(* IEC 61131-3 sources: std_i2980_v2.06_cp053/Source/IMM/ieccontrol/HeatingGeneral (part 2) *)

//*********************************************************************************************
// Temperature optimization
//*********************************************************************************************
//checking startconditions for temp optimization
fbRTrigRunOptimization(CLK := sv_bRunOptimization);
IF (fbRTrigRunOptimization.Q) THEN
   aCheckOptimizeStartConditions(nOptState := enOPOState);
END_IF;

IF enOPOState = enOPOState_StableFirst OR enOPOState = enOPOState_StableSecond THEN
   bGroupStable := TRUE;
   FOR i := 1 TO miNumberOfZones DO
      IF sv_ZoneArray[i].DataRetain^.bUsed THEN
         //ignore zones which are not used
         bGroupStable := bGroupStable AND (sv_ZoneArray[i].Data^.Stable = KCTRL_Stable_OK);
      END_IF;
   END_FOR;

   IF bGroupStable AND enOPOState = enOPOState_StableFirst THEN
      i := 0;
      WHILE 2*i + 1 <= miNumberOfZones DO
         IF sv_ZoneArray[2*i + 1].Data^.bSensorOK AND
            sv_ZoneArray[2*i + 1].Data^.bOutputOK AND
            sv_ZoneArray[2*i + 1].DataRetain^.SensorTypeVis <> KHW_TempSensor_none AND
            sv_ZoneArray[2*i + 1].DataRetain^.Param.opMode <> KAPPL_TempOpMode_Cooling THEN
            sv_ZoneArray[2*i + 1].Data^.bOptimize := TRUE;
            sv_ZoneArray[2*i + 1].Data^.bOptiOperatingPoint := TRUE;
         END_IF;
      i := i + 1;
      END_WHILE;
      enOPOState := enOPOState_RunFirst;
   ELSIF bGroupStable AND enOPOState = enOPOState_StableSecond THEN
      // second part of operation point calibration has to be used
      i := 1;
      WHILE 2*i <= miNumberOfZones DO
         IF sv_ZoneArray[2*i].Data^.bSensorOK AND
            sv_ZoneArray[2*i].Data^.bOutputOK AND
            sv_ZoneArray[2*i].DataRetain^.SensorTypeVis <> KHW_TempSensor_none AND
            sv_ZoneArray[2*i].DataRetain^.Param.opMode <> KAPPL_TempOpMode_Cooling THEN
            sv_ZoneArray[2*i].Data^.bOptimize := TRUE;
            sv_ZoneArray[2*i].Data^.bOptiOperatingPoint := TRUE;
         END_IF;
      i := i + 1;
      END_WHILE;
      enOPOState := enOPOState_None;
   END_IF;

END_IF;

fbRTrigOptimizationActive(CLK := sv_bOptimizationActive);//optimization started detection
fbFTrigOptimizationActive(CLK := sv_bOptimizationActive);//optimization ready detection
fbFTrigOptimizationInterrupt(CLK:= sv_bRunOptimization);//optimization stopped manually
bGroupOn := bHeatingOn;
IF fbFTrigOptimizationActive.Q THEN
   FOR i := 1 TO miNumberOfZones DO
      sv_ZoneArray[i].Data^.bOptimize := FALSE;
      // check parameters valid
      aCheckPIDParameter(iIndex2Check := i,
                         iMaxNoZones := miNumberOfZones);
   END_FOR;
   IF enOPOState = enOPOState_None THEN
      // optimization ready
      sv_bRunOptimization := FALSE;
   ELSE
      IF miNumberOfZones > 1 THEN
         enOPOState := enOPOState_StableSecond;
      ELSE  // only 1 zone optimization ready
         enOPOState := enOPOState_None;
         sv_bRunOptimization := FALSE;
      END_IF;
   END_IF;
END_IF;

//*********************************************************************************************
// Calculate set value for normal and group heating
//*********************************************************************************************
IF bHeatingOn THEN
   //call group block

   // Find Min/Max from ActValues for starting with temperatures
   // in toleranceband, checking whether the temperatures are
   // stabil relatively to each other
   MinActValues := 1000.0;
   MaxActValues := 0.0;
   FOR i := 1 TO miNumberOfZones DO
      IF sv_ZoneArray[i].Data^.bSensorOK THEN
        IF sv_ZoneArray[i].Data^.prActTemp^ < MinActValues
            AND sv_ZoneArray[i].DataRetain^.Param.bZoneUsedForGroupHeating THEN
            MinActValues := sv_ZoneArray[i].Data^.prActTemp^;
            iIndexMinZone := i;
        END_IF;
        IF sv_ZoneArray[i].Data^.prActTemp^ > MaxActValues
            AND sv_ZoneArray[i].DataRetain^.Param.bZoneUsedForGroupHeating THEN
            MaxActValues := sv_ZoneArray[i].Data^.prActTemp^;
        END_IF;
      END_IF;
   END_FOR;

   // Heating up to same temperature
   // StartGroupHeating
   IF GroupHeatingStatus = 1 THEN
      IF (((MaxActValues - MinActValues)> sv_rTolBetweenZones * 0.5) OR
          (CountStartGroupHeating < ObservationFactor)) THEN
         // Checking stability
         IF (MaxActValues - MinActValues) <= sv_rTolBetweenZones * 0.5 THEN
            CountStartGroupHeating := CountStartGroupHeating + 1;
            iIndexMinZone := 0; // no zone has set value from vis
         ELSE
            CountStartGroupHeating := 1;
         END_IF;
         IF (SetStartTemperatureGroupHeating < MinActValues) THEN
            SetStartTemperatureGroupHeating := MinActValues;
         END_IF;
         // Set the SetValues and switching of the GroupHeating temporary
         fbHeatingGroup.GroupHeating := FALSE;
          FOR i := 1 TO miNumberOfZones DO
             fbHeatingGroup.ZoneUsed[i] := sv_ZoneArray[i].DataRetain^.Param.bZoneUsedForGroupHeating;
             IF NOT sv_bKeepWarmActive THEN
                // Heating to the hotest Zonetemperature
                fbHeatingGroup.SetValues[i] := SetStartTemperatureGroupHeating;
             ELSE
                fbHeatingGroup.SetValues[i] := sv_ZoneArray[i].DataRetain^.rStandbyTempVis;
             END_IF;
             IF sv_ZoneArray[i].Data^.bSensorOK THEN
                fbHeatingGroup.ActValues[i] := sv_ZoneArray[i].Data^.prActTemp^;
             END_IF;
          END_FOR;
      ELSE
      fbHeatingGroup.GroupHeating := TRUE;
      GroupHeatingStatus := 2;
      END_IF;
   END_IF; // END GroupHeatingStatus = 1
   IF NOT (GroupHeatingStatus = 1) THEN
      FOR i := 1 TO miNumberOfZones DO
         fbHeatingGroup.ZoneUsed[i] := sv_ZoneArray[i].DataRetain^.Param.bZoneUsedForGroupHeating;
         IF NOT sv_bKeepWarmActive THEN
            IF sv_ZoneArray[i].Data^.bUseIncTemperature THEN
               fbHeatingGroup.SetValues[i] := sv_ZoneArray[i].DataRetain^.rSetValVis + sv_rIncTemperature;
            ELSE
               fbHeatingGroup.SetValues[i] := sv_ZoneArray[i].DataRetain^.rSetValVis;
            END_IF;
         ELSE
            fbHeatingGroup.SetValues[i] := sv_ZoneArray[i].DataRetain^.rStandbyTempVis;
         END_IF;
         IF sv_ZoneArray[i].Data^.bSensorOK THEN
            fbHeatingGroup.ActValues[i] := sv_ZoneArray[i].Data^.prActTemp^;
         END_IF;
      END_FOR;
      IF GroupHeatingStatus = 2 THEN
         IF (MaxActValues - MinActValues) > sv_rTolBetweenZones THEN
            bOutOfTol := TRUE;
         END_IF;
         bReadyGroupHeating := TRUE;
         FOR i := 1 TO miNumberOfZones DO
            //groupheating ignored for zones where no TI-sensor or zone not useful for GH (setter, measure mode)
            IF sv_ZoneArray[i].Data^.bSensorOK AND sv_ZoneArray[i].DataRetain^.Param.bZoneUsedForGroupHeating THEN
                IF ABS(sv_ZoneArray[i].Data^.prActTemp^-MinSetValues) > sv_rTolBetweenZones * 0.5 THEN
                    bReadyGroupHeating := FALSE;
                    EXIT;
                END_IF;
            END_IF;
         END_FOR;
         IF bReadyGroupHeating THEN
            GroupHeatingStatus := 0;
            fbHeatingGroup.GroupHeating := FALSE;
         END_IF;
      END_IF;
   END_IF;
   fbHeatingGroup(ReParam := FALSE,
                  bHeatingOn := bHeatingOn);
END_IF; //END bHeatingOn (call group block)

//*********************************************************************************************
// Set calculated set value for each zone
//*********************************************************************************************
fbRTrigSetValChanged(CLK:= fbHeatingGroup.bAnyValueChanged);
IF NOT sv_bOptimizationActive THEN
   //normal operation, copy values from group - block
   FOR i := 1 TO miNumberOfZones DO
      IF ((NOT bHeatingOn) AND (sv_ZoneArray[i].DataRetain^.Param.opMode = KAPPL_TempOpMode_Cooling)) THEN
         sv_ZoneArray[i].Data^.PWMFactor := 1.0;
         sv_ZoneArray[i].Data^.rSetVal   := sv_ZoneArray[i].DataRetain^.rSetValVis;
      ELSE
         sv_ZoneArray[i].Data^.PWMFactor := fbHeatingGroup.PWMFactor[i];
         sv_ZoneArray[i].Data^.rSetVal   := fbHeatingGroup.OutputValues[i];
      END_IF;
   END_FOR;
ELSE // optimization, use value from visualisation
    FOR i := 1 TO miNumberOfZones DO
      sv_ZoneArray[i].Data^.PWMFactor := 1.0;
      sv_ZoneArray[i].Data^.rSetVal :=  sv_ZoneArray[i].DataRetain^.rSetValVis;
   END_FOR;
END_IF;

//*********************************************************************************************
// Check state of optimization
//*********************************************************************************************
//optimization interrupted manually
IF (((fbFTrigOptimizationInterrupt.Q OR fbFTrigHeatingOn.Q) AND
     (sv_bOptimizationActive OR (enOPOState <> enOPOState_None))) OR
    (fbFTrigOptimizationInterrupt.Q AND NOT bHeatingOn AND NOT
     (sv_bOptimizationActive OR (enOPOState <> enOPOState_None)))) THEN
   FOR i := 1 TO miNumberOfZones DO
      sv_ZoneArray[i].Data^.bOptimize := FALSE;
   END_FOR;
   sv_bRunOptimization := FALSE;
END_IF;

bOptimizinActive := FALSE;
FOR i := 1 TO miNumberOfZones DO
   //check if any zone is optimizing
   IF sv_ZoneArray[i].Data^.bIsOptimizing THEN
      bOptimizinActive := TRUE;
      EXIT;
   END_IF;
END_FOR;

sv_bOptimizationActive := bOptimizinActive;

//*********************************************************************************************
// Failure control and Output
//*********************************************************************************************

//also consider zones which are not handled in groupheating
aCheckNonGroupHeatingZones();
bOtherZonesReady := aCheckNonGroupHeatingZones.bAllZonesInTolerance;

//Minutes to seconds
sv_dTempOkTimeSet :=  LINT_TO_TIME(REAL_TO_LINT(sv_rTempOkTimeSet * 60.0 * 1000.0 * 1000.0));
fbTonTempOkTime(IN := (fbHeatingGroup.AllZonesReady AND bHeatingOn AND bOtherZonesReady),
                PT := sv_dTempOkTimeSet);
sv_dTempOkTimeAct := fbTonTempOkTime.ET;
sv_rTempOkTimeAct := LINT_TO_REAL(TIME_TO_LINT(sv_dTempOkTimeAct))/(60.0 * 1000.0 * 1000.0);
bGroupTempOK := fbTonTempOkTime.Q;
fbFTrigGroupTempOK(CLK := bGroupTempOK);
fbRTrigGroupTempOK(CLK := bGroupTempOK);

// Check state of heating and set/reset alarm
// Folowing states are possible
// Heat Up Active
// Keep Warm Active
// Cool Prevent Time is running (Temperature first time in tolerance)
// None: Heating off, heating stable in operating point
IF sv_bKeepWarmActive AND NOT bKeepWarmActive THEN
    bKeepWarmActive := TRUE;
    SET_ALARM (Name := erKeepWarmActive,
                SubID1 := sv_DeviceId.CompId,
                SubID2 := sv_DeviceId.IndexId);
END_IF;
IF bKeepWarmActive AND NOT sv_bKeepWarmActive THEN
    bKeepWarmActive := FALSE;
    RESET_ALARM (Name := erKeepWarmActive,
                SubID1 := sv_DeviceId.CompId,
                SubID2 := sv_DeviceId.IndexId);
END_IF;

IF bCoolPrevent AND (bKeepWarmActive OR NOT bHeatingOn OR bGroupTempOK OR fbRTrigSetValChanged.Q) THEN
    bCoolPrevent := FALSE;
    RESET_ALARM (Name := erCoolingPrevent,
                SubID1 := sv_DeviceId.CompId,
                SubID2 := sv_DeviceId.IndexId);
END_IF;
IF NOT bCoolPrevent AND NOT bKeepWarmActive AND bHeatingOn AND NOT bGroupTempOK AND fbHeatingGroup.AllZonesReady AND bOtherZonesReady THEN
    bCoolPrevent := TRUE;
    SET_ALARM (Name := erCoolingPrevent,
                SubID1 := sv_DeviceId.CompId,
                SubID2 := sv_DeviceId.IndexId);
END_IF;

IF NOT bKeepWarmActive AND NOT mbHeatUp AND NOT bCoolPrevent AND(
    (fbRTrigHeatingOn.Q AND NOT bGroupTempOK) OR
    (bHeatingOn AND fbRTrigSetValChanged.Q AND NOT bGroupTempOK) OR
    ((sv_bGroupHeating AND fbRTrigHeatingOn.Q) OR (fbRTrigGroupHeating.Q AND bHeatingOn)) OR
    (fbFTrigOptimizationActive.Q AND NOT fbHeatingGroup.AllZonesReady)
    )THEN
    mbHeatUp := TRUE;
    SET_ALARM (Name := erHeatupActive,
                SubID1 := sv_DeviceId.CompId,
                SubID2 := sv_DeviceId.IndexId);
END_IF;
IF mbHeatUp AND (bKeepWarmActive OR bCoolPrevent OR NOT bHeatingOn OR bGroupTempOK OR fbHeatingGroup.AllZonesReady) THEN
   mbHeatUp := FALSE;
   RESET_ALARM (Name := erHeatupActive,
                SubID1 := sv_DeviceId.CompId,
                SubID2 := sv_DeviceId.IndexId);
END_IF;

(*      tolerance supervision       *)
IF fbFTrigGroupTempOK.Q THEN
    bOutOfTolerance := TRUE;
END_IF;
IF fbRTrigGroupTempOK.Q THEN
    bOutOfTolerance := FALSE;
END_IF;
IF ((bOutOfTolerance OR fbRTrigGroupTempOK.Q) AND
    (NOT (mbHeatUp OR bCoolPrevent OR sv_bRunOptimization)) OR (NOT bHeatingOn)) THEN

    FOR i := 1 TO miNumberOfZones DO
        (* searching for the zones which are out ouf tol *)
        IF (sv_ZoneArray[i].Data^.bToleranceError AND (NOT ToleranceAlarm[i])) AND
           (bHeatingOn AND (NOT (mbHeatUp OR bCoolPrevent))) THEN
            (* setting tolerance error *)
            IF ((sv_ZoneArray[i].Data^.bEmgOperation AND sv_OperationMode >= nHalfAutomatic)) OR
                bKeepWarmActive OR bGroupActive THEN
               ; // no Alarm Emergency operation mode
            ELSE
               ToleranceAlarm[i] := TRUE;
               SET_ALARM (Name := erZoneOutOfTol,
                        SubID1 := sv_DeviceId.CompId,
                        SubID2 := sv_DeviceId.IndexId,
                        SubID3 := i);
           END_IF;
        END_IF;

        IF  (NOT sv_ZoneArray[i].Data^.bToleranceError AND ToleranceAlarm[i]) OR
            (NOT bHeatingOn AND ToleranceAlarm[i]) OR (NOT sv_ZoneArray[i].DataRetain^.bUsed)  THEN

            ToleranceAlarm[i] := FALSE;
            RESET_ALARM (Name := erZoneOutOfTol,
                    SubID1 := sv_DeviceId.CompId,
                    SubID2 := sv_DeviceId.IndexId,
                    SubID3 := i);
        END_IF;
    END_FOR;
END_IF;

// set/reset status message during temp.optimization
IF fbRTrigOptimizationActive.Q THEN
    SET_ALARM (Name := erOptimizationActive,
              SubID1 := sv_DeviceId.CompId,
              SubID2 := sv_DeviceId.IndexId);
END_IF;

IF fbFTrigOptimizationActive.Q THEN
    RESET_ALARM (Name := erOptimizationActive,
                SubID1 := sv_DeviceId.CompId,
                SubID2 := sv_DeviceId.IndexId);
END_IF;

fbRTrigOutOfTol(CLK:=bOutOfTol);
IF fbRTrigOutOfTol.Q THEN
   SET_ALARM (Name := erOutOfTol,
              SubID1 := sv_DeviceId.CompId,
              SubID2 := sv_DeviceId.IndexId);
END_IF;

bGroupActive := (GroupHeatingStatus > 0);

@END_Body

@@@BEG_Comment@@@
@TL(0)

@@@END_Comment@@@

@BEG_Body
@TL(9)
(**************************************** WARNING ********************************************
 *** The KEBA Kemro K2 System including software is not intended for safety control tasks! ***
 ***                       For further information see Comment tab!                        ***
 *********************************************************************************************)

//reparam Group
mbInit := FALSE;
sv_bReParamGroup := FALSE;

@END_Body

@@@BEG_Comment@@@
@TL(0)

@@@END_Comment@@@

@BEG_Body
@TL(7)
(**************************************** WARNING ********************************************
 *** The KEBA Kemro K2 System including software is not intended for safety control tasks! ***
 ***                       For further information see Comment tab!                        ***
 *********************************************************************************************)

START_PROCESS_ALGORITHM(paCheckNumberOfZones);

@END_Body

@@@BEG_Comment@@@
@TL(0)

@@@END_Comment@@@

@BEG_Body
@TL(52)
(**************************************** WARNING ********************************************
 *** The KEBA Kemro K2 System including software is not intended for safety control tasks! ***
 ***                       For further information see Comment tab!                        ***
 *********************************************************************************************)

IF mbInitDone THEN

   FOR i := 1 TO sv_iMaxNumberOfZones DO

      IF i <= sv_iZonesAvailable AND i <= sv_iNumberOfZones AND sv_ZoneArray[i].bLinked THEN
            //tell the zone that it will be used
            //set counter for aRun to prevent from nullpointerexception if wrong mold data was loaded (sv_iNumberOfZones > sv_iZonesAvailable)
            miNumberOfZones := i;
            // Dont set value higher than max allowed temperature
            sv_ZoneArray[i].Data^.bOutputNotAllowed := FALSE;
            sv_ZoneArray[i].DataRetain^.rSetValVis := MIN(sv_rMaxTemperature, sv_ZoneArray[i].DataRetain^.rSetValVis);
            // heating nozzle zone is always used
            IF NOT (sv_ZoneArray[i].DataRetain^.bIsHotrunner OR sv_ZoneArray[i].DataRetain^.ZoneType = enZoneTypeBlock) THEN
               sv_ZoneArray[i].DataRetain^.bUsed := TRUE;
            END_IF;
      ELSIF sv_ZoneArray[i].bLinked THEN
            sv_ZoneArray[i].DataRetain^.bUsed := FALSE;
      END_IF;

      IF i > sv_iZonesAvailable AND i <= sv_iNumberOfZones THEN
         //zone is used but Hardware is not OK -> error
            SET_ALARM(Name := erZoneNotAvailable,
                      SubID1 := sv_DeviceId.CompId,
                      SubID2 := sv_DeviceId.IndexId,
                      SubID3 := i);
      END_IF;

      IF  i > sv_iNumberOfZones AND i <= iNumberOfZonesOld AND i > sv_iZonesAvailable THEN
         //reset alarm if sv_iNumberOfZones has been reduced
         RESET_ALARM(Name := erZoneNotAvailable,
                     SubID1 := sv_DeviceId.CompId,
                     SubID2 := sv_DeviceId.IndexId,
                     SubID3 := i);
         IF (sv_ZoneArray[i].bLinked) AND
            NOT (sv_ZoneArray[i].DataRetain^.bIsHotrunner OR sv_ZoneArray[i].DataRetain^.ZoneType = enZoneTypeBlock) THEN
            sv_ZoneArray[i].DataRetain^.bUsed := TRUE;
         END_IF;

      END_IF;
   END_FOR;
   STOP_PROCESS_ALGORITHM();
END_IF;

iNumberOfZonesOld := sv_iNumberOfZones;

@END_Body

@@@BEG_Comment@@@
@TL(0)

@@@END_Comment@@@

@BEG_Body
@TL(7)
// After max temperature changed, dont allow higher set values
FOR i := 1 TO miNumberOfZones DO
    IF sv_ZoneArray[i].DataRetain^.rSetValVis > sv_rMaxTemperature THEN
       sv_ZoneArray[i].DataRetain^.rSetValVis := sv_rMaxTemperature;
    END_IF;
END_FOR;

@END_Body

@@@BEG_Comment@@@
@TL(0)

@@@END_Comment@@@

@BEG_Body
@TL(18)
IF sv_bUndoChangeHeatingParams THEN
   IF NOT mbInitDone THEN
      sv_bUndoChangeHeatingParams := FALSE;
      RETURN;
   END_IF;
   FOR i := 1 TO miNumberOfZones DO
      IF sv_ZoneArray[i].DataRetain^.Param.bOldPIDAvailable THEN
         sv_ZoneArray[i].DataRetain^.Param.pidParam := sv_ZoneArray[i].DataRetain^.Param.pidParamLastOpt;
         sv_bUsePidOP := FALSE;
         sv_bReParamGroup := TRUE;
         sv_ZoneArray[i].DataRetain^.Param.bOldPIDAvailable := FALSE;
      END_IF;
   END_FOR;
   //reparam tempgroup
   // reset sv
   sv_bUndoChangeHeatingParams := FALSE;
END_IF;

@END_Body

@@@BEG_Comment@@@
@TL(0)

@@@END_Comment@@@

@BEG_Body
@TL(7)
(**************************************** WARNING ********************************************
 *** The KEBA Kemro K2 System including software is not intended for safety control tasks! ***
 ***                       For further information see Comment tab!                        ***
 *********************************************************************************************)

rActTemp := sv_ZoneArray[miLeadingZone].Data^.prActTemp^;

@END_Body

@@@BEG_Comment@@@
@TL(0)

@@@END_Comment@@@
@END_Body

@END_Contents

(* ---- ABHopperCooling.pu ---- *)
(*
This Algorithm Block is responsible for
  - hopper temp. supervision
  - hopper cooling

*)

IMPORT_OVER_LISTFILE
 KSWO_AddVariable
, SET_ALARM
, RESET_ALARM
, FGetHWPath
, GET_MY_FU_NAME
, KHW_TempSensor
, tsDeviceId
, KSWO_Status
, R_TRIG

END_IMPORT

ALGORITHM_BLOCK ABHopperCooling #DUMMY_EDIT_BLOCK

SYSTEM_VAR
 do_HopperCooler : BOOL;
 ti_HopperTemp : REAL;
 ti_HopperTemp_sensor : KHW_TempSensor;
 ti_HopperTemp_stat : BOOL;
 sv_rTempStartCooling : REAL (* start cooling at this temperature *);
 sv_rTempStopCooling : REAL (* stop cooling at this temperature *);
 sv_rWarnTemp : REAL (* a warning is displayed if hopper temperature increases this value *);
 sv_rAlarmTemp : REAL (* an alarm is displayed if hopper temperature increases this value *);
 sv_HopperTempSensorType : KHW_TempSensor (* sensor type *);
 sv_rHopperTempHysteresis : REAL;
 sv_DeviceId : tsDeviceId;
END_VAR

SYSTEM_OBJECT
 PU_Task_7 : TASK;
 TaskSlow : TASK;
 erHopperTempWarning : ALARM;
 erHopperTempTooHigh : ALARM;
 erHopperTempSensor : ALARM;
END_OBJECT

VAR
 mbSensorError : BOOL;
 msHWPath : STRING(255);
 mpbSensorState : REFTO BOOL;
END_VAR

ALGORITHM aSensorState

#BEGIN_EDIT_BLOCK
(**************************************** WARNING ********************************************
 *** The KEBA Kemro K2 System including software is not intended for safety control tasks! ***
 ***                       For further information see Comment tab!                        ***
 *********************************************************************************************)

mbSensorError := ti_HopperTemp_stat;

IF mbSensorError THEN

   //reset digital output for cooling in case of sensor error
   IF IS_LINKED(do_HopperCooler) THEN
      do_HopperCooler := FALSE;
   END_IF;

   SET_ALARM(Name := erHopperTempSensor,
             SubID1 := sv_DeviceId.CompId,
             SubID2 := sv_DeviceId.IndexId,
             Param1 := msHWPath);
ELSE
   RESET_ALARM(Name := erHopperTempSensor,
               SubID1 := sv_DeviceId.CompId,
               SubID2 := sv_DeviceId.IndexId);
END_IF;

;#END_EDIT_BLOCK END_ALGORITHM

(*
Check which Inputs and Outputs are available and start according process algorithms
*)

PROCESS_ALGORITHM paInit ON TaskSlow AUTOSTART

VAR
 swoState : KSWO_Status;
END_VAR
#BEGIN_EDIT_BLOCK
(**************************************** WARNING ********************************************
 *** The KEBA Kemro K2 System including software is not intended for safety control tasks! ***
 ***                       For further information see Comment tab!                        ***
 *********************************************************************************************)

IF IS_LINKED(ti_HopperTemp) AND IS_LINKED(ti_HopperTemp_stat) THEN

   ti_HopperTemp_sensor := sv_HopperTempSensorType;

   msHWPath := FGetHWPath(CONCAT(GET_MY_FU_NAME(),'.ti_HopperTemp'), TRUE);
   mpbSensorState := @ti_HopperTemp_stat;

   aSensorState();

   swoState := KSWO_AddVariable( Task := TaskSlow,
                                 Name := 'HopperTemperature',
                                 Variable := ti_HopperTemp);

   //start supervision of hopper temperature
   START_PROCESS_ALGORITHM(paHopperTempSupervision);

   IF IS_LINKED(do_HopperCooler) THEN
      //start algorithm for hopper cooling
      START_PROCESS_ALGORITHM(paHopperCooler);
   END_IF;
END_IF;

STOP_PROCESS_ALGORITHM();

;#END_EDIT_BLOCK END_ALGORITHM

(*
In this algorithm the supervision of the material temperature is done.
If actual material temp is higher than the alarm temperature an alarm is set.
If actual material temperature is lower than alarm temp -5° the alarm is resetted.
Setting the material temp high - alarm causes a stop of the motor!
Switching on the motor is only possible if the material temperature is ok again.
*)

PROCESS_ALGORITHM paHopperTempSupervision ON TaskSlow

VAR
 fbRTrigWarningTemp : R_TRIG;
 fbRTrigAlarmTemp : R_TRIG;
 fbRTrigWarningTempOk : R_TRIG;
 fbRTrigAlarmTempOk : R_TRIG;
END_VAR
#BEGIN_EDIT_BLOCK
(**************************************** WARNING ********************************************
 *** The KEBA Kemro K2 System including software is not intended for safety control tasks! ***
 ***                       For further information see Comment tab!                        ***
 *********************************************************************************************)

fbRTrigWarningTemp(CLK := (ti_HopperTemp > sv_rWarnTemp));
fbRTrigWarningTempOk(CLK := (ti_HopperTemp < (sv_rWarnTemp - sv_rHopperTempHysteresis)));

fbRTrigAlarmTemp(CLK := (ti_HopperTemp > sv_rAlarmTemp));
fbRTrigAlarmTempOk(CLK := (ti_HopperTemp < (sv_rAlarmTemp - sv_rHopperTempHysteresis)));

IF fbRTrigWarningTemp.Q THEN
   //set alarm if warning temp is exceeded
   SET_ALARM (Name := erHopperTempWarning,
              SubID1 := sv_DeviceId.CompId,
              SubID2 := sv_DeviceId.IndexId);
END_IF;

IF fbRTrigWarningTempOk.Q THEN
   //reset alarm if temp is ok again
   RESET_ALARM (Name := erHopperTempWarning,
                SubID1 := sv_DeviceId.CompId,
                SubID2 := sv_DeviceId.IndexId);
END_IF;

IF fbRTrigAlarmTemp.Q THEN
   //set alarm if alarm temp is exceeded
   SET_ALARM (Name := erHopperTempTooHigh,
              SubID1 := sv_DeviceId.CompId,
              SubID2 := sv_DeviceId.IndexId);
END_IF;

IF fbRTrigAlarmTempOk.Q THEN
   //set alarm if temp is ok again
   RESET_ALARM (Name := erHopperTempTooHigh,
                SubID1 := sv_DeviceId.CompId,
                SubID2 := sv_DeviceId.IndexId);
END_IF;

;#END_EDIT_BLOCK END_ALGORITHM

(*
If a digital output for hopper cooling is available it will be set if the
actual material temperature is higher than start cooling temperature.
The DO will be resetted after the actual temperature is lower than stop cooling temperature.
In case of a sensor error the DO will also be resetted.
*)

PROCESS_ALGORITHM paHopperCooler ON TaskSlow

VAR
 fbRTrigStartCooling : R_TRIG;
 fbRTrigStopCooling : R_TRIG;
END_VAR
#BEGIN_EDIT_BLOCK
(**************************************** WARNING ********************************************
 *** The KEBA Kemro K2 System including software is not intended for safety control tasks! ***
 ***                       For further information see Comment tab!                        ***
 *********************************************************************************************)

fbRTrigStartCooling(CLK := (ti_HopperTemp > sv_rTempStartCooling));
fbRTrigStopCooling(CLK := (ti_HopperTemp < sv_rTempStopCooling));

IF fbRTrigStartCooling.Q AND NOT mbSensorError THEN
   //set digital output for cooling
   do_HopperCooler := TRUE;
END_IF;

IF fbRTrigStopCooling.Q THEN
   //reset digital output for cooling
   do_HopperCooler := FALSE;
END_IF;

;#END_EDIT_BLOCK END_ALGORITHM

POSTUPDATE_ALGORITHM pSensorTypeChanged ON PU_Task_7 WITH sv_HopperTempSensorType

#BEGIN_EDIT_BLOCK
(**************************************** WARNING ********************************************
 *** The KEBA Kemro K2 System including software is not intended for safety control tasks! ***
 ***                       For further information see Comment tab!                        ***
 *********************************************************************************************)

//copy selected sensor type
ti_HopperTemp_sensor := sv_HopperTempSensorType;

;#END_EDIT_BLOCK END_ALGORITHM

(*
react on changes of material temp sensor state
*)

POSTUPDATE_ALGORITHM pSensorStateChanged ON PU_Task_7 WITH mpbSensorState^

#BEGIN_EDIT_BLOCK
(**************************************** WARNING ********************************************
 *** The KEBA Kemro K2 System including software is not intended for safety control tasks! ***
 ***                       For further information see Comment tab!                        ***
 *********************************************************************************************)

aSensorState();

;#END_EDIT_BLOCK END_ALGORITHM

END_ALGORITHM_BLOCK

#END_OF_IEC_PART

@Puma @IecEditor 6 68 @Pou 25
@@@BEG_Comment@@@
This Algorithm Block is responsible for
  - hopper temp. supervision
  - hopper cooling

@@@END_Comment@@@

@BEG_Contents

@BEG_Func
@RT(17)FuncTreeContainer
5
@Var @RT(16)KSWO_AddVariable @RT(0) @T @T @DERIVED 0 @F @RT(22)KEBA_STANDARD_FUNCTION @F
@T
@BEG_Attrib
0 @RT(0) @RT(0)
@END_Attrib
1 1 @F @F @F @F

@Var @RT(9)SET_ALARM @RT(0) @T @T @DERIVED 0 @F @RT(23)KEBA_STANDARD_PROCEDURE @F
@T
@BEG_Attrib
0 @RT(0) @RT(0)
@END_Attrib
1 1 @F @F @F @F

@Var @RT(11)RESET_ALARM @RT(0) @T @T @DERIVED 0 @F @RT(23)KEBA_STANDARD_PROCEDURE @F
@T
@BEG_Attrib
0 @RT(0) @RT(0)
@END_Attrib
1 1 @F @F @F @F

@Var @RT(10)FGetHWPath @RT(0) @T @T @DERIVED 0 @F @RT(8)FUNCTION @F
@T
@BEG_Attrib
0 @RT(0) @RT(0)
@END_Attrib
1 1 @F @F @F @F

@Var @RT(14)GET_MY_FU_NAME @RT(0) @T @T @DERIVED 0 @F @RT(22)KEBA_STANDARD_FUNCTION @F
@T
@BEG_Attrib
0 @RT(0) @RT(0)
@END_Attrib
1 1 @F @F @F @F

@END_Func

@BEG_Const
@RT(18)ConstTreeContainer
0
@END_Const

@BEG_Export

@BEG_Kind
@ALGORITHM_BLOCK @RT(15)ABHopperCooling @STRUCTURED_TEXT
@RT(0) @RT(0) @RT(0)
@END_Kind

@BEG_Dcl
@RT(16)DclTreeContainer
19
@Var @RT(15)do_HopperCooler @RT(0) @T @F @DT @RT(4)BOOL @RT(0) @T @T @BASIC 0 @F
@F @F
@T
@BEG_Attrib
3 @RT(0) @RT(0) @RT(0)
@END_Attrib
1 8 @F @F @F @F

@Var @RT(13)ti_HopperTemp @RT(0) @T @F @DT @RT(4)REAL @RT(0) @T @T @BASIC 0 @F
@F @F
@T
@BEG_Attrib
3 @RT(0) @RT(0) @RT(0)
@END_Attrib
1 8 @F @F @F @F

@Var @RT(20)ti_HopperTemp_sensor @RT(0) @T @T @DERIVED 0 @T @T @DT @RT(14)KHW_TempSensor @RT(0) @T @T @UNKNOWN 0 @F
@F @F
@T
@BEG_Attrib
3 @RT(0) @RT(0) @RT(0)
@END_Attrib
1 8 @F @F @F @F

@Var @RT(18)ti_HopperTemp_stat @RT(0) @T @F @DT @RT(4)BOOL @RT(0) @T @T @BASIC 0 @F
@F @F
@T
@BEG_Attrib
3 @RT(0) @RT(0) @RT(0)
@END_Attrib
1 8 @F @F @F @F

@Var @RT(20)sv_rTempStartCooling @RT(0) @T @F @DT @RT(4)REAL @RT(0) @T @T @BASIC 0 @F
@F @F
@T
@BEG_Attrib
3 @RT(0) @RT(33)start cooling at this temperature @RT(0)
@END_Attrib
1 8 @F @F @F @F

@Var @RT(19)sv_rTempStopCooling @RT(0) @T @F @DT @RT(4)REAL @RT(0) @T @T @BASIC 0 @F
@F @F
@T
@BEG_Attrib
3 @RT(0) @RT(32)stop cooling at this temperature @RT(0)
@END_Attrib
1 8 @F @F @F @F

@Var @RT(12)sv_rWarnTemp @RT(0) @T @F @DT @RT(4)REAL @RT(0) @T @T @BASIC 0 @F
@F @F
@T
@BEG_Attrib
3 @RT(0) @RT(65)a warning is displayed if hopper temperature increases this value @RT(0)
@END_Attrib
1 8 @F @F @F @F

@Var @RT(13)sv_rAlarmTemp @RT(0) @T @F @DT @RT(4)REAL @RT(0) @T @T @BASIC 0 @F
@F @F
@T
@BEG_Attrib
3 @RT(0) @RT(64)an alarm is displayed if hopper temperature increases this value @RT(0)
@END_Attrib
1 8 @F @F @F @F

@Var @RT(23)sv_HopperTempSensorType @RT(0) @T @T @DERIVED 0 @T @T @DT @RT(14)KHW_TempSensor @RT(0) @T @T @UNKNOWN 0 @F
@F @F
@T
@BEG_Attrib
3 @RT(0) @RT(11)sensor type @RT(0)
@END_Attrib
1 8 @F @F @F @F

@Var @RT(9)PU_Task_7 @RT(0) @T @F @DT @RT(4)TASK @RT(0) @T @T @BASIC 0 @F
@F @F
@T
@BEG_Attrib
3 @RT(0) @RT(0) @RT(0)
@END_Attrib
1 7 @F @F @F @F

@Var @RT(8)TaskSlow @RT(0) @T @F @DT @RT(4)TASK @RT(0) @T @T @BASIC 0 @F
@F @F
@T
@BEG_Attrib
3 @RT(0) @RT(0) @RT(0)
@END_Attrib
1 7 @F @F @F @F

@Var @RT(19)erHopperTempWarning @RT(0) @T @F @DT @RT(5)ALARM @RT(0) @T @T @BASIC 0 @F
@F @F
@T
@BEG_Attrib
3 @RT(0) @RT(0) @RT(0)
@END_Attrib
1 7 @F @F @F @F

@Var @RT(19)erHopperTempTooHigh @RT(0) @T @F @DT @RT(5)ALARM @RT(0) @T @T @BASIC 0 @F
@F @F
@T
@BEG_Attrib
3 @RT(0) @RT(0) @RT(0)
@END_Attrib
1 7 @F @F @F @F

@Var @RT(18)erHopperTempSensor @RT(0) @T @F @DT @RT(5)ALARM @RT(0) @T @T @BASIC 0 @F
@F @F
@T
@BEG_Attrib
3 @RT(0) @RT(0) @RT(0)
@END_Attrib
1 7 @F @F @F @F

@Var @RT(13)mbSensorError @RT(0) @T @F @DT @RT(4)BOOL @RT(0) @T @T @BASIC 0 @F
@F @F
@T
@BEG_Attrib
3 @RT(0) @RT(0) @RT(0)
@END_Attrib
1 0 @F @F @F @F

@Var @RT(24)sv_rHopperTempHysteresis @RT(0) @T @F @DT @RT(4)REAL @RT(0) @T @T @BASIC 0 @F
@F @F
@T
@BEG_Attrib
3 @RT(0) @RT(0) @RT(0)
@END_Attrib
1 8 @F @F @F @F

@Var @RT(8)msHWPath @RT(0) @T @F @DT @RT(11)STRING(255) @RT(0) @T @T @STRING 0 @F @RT(3)255 @F
@F @F
@T
@BEG_Attrib
3 @RT(0) @RT(0) @RT(0)
@END_Attrib
1 0 @F @F @F @F

@Var @RT(14)mpbSensorState @RT(0) @T @T @REFTO 0 @T @DT @RT(4)BOOL @RT(0) @T @T @BASIC 0 @F
@F @F
@T
@BEG_Attrib
3 @RT(0) @RT(0) @RT(0)
@END_Attrib
1 0 @F @F @F @F

@Var @RT(11)sv_DeviceId @RT(0) @T @T @DERIVED 0 @F @RT(10)tsDeviceId @F
@T
@BEG_Attrib
3 @RT(0) @RT(0) @RT(0)
@END_Attrib
1 8 @F @F @F @F

@END_Dcl

@END_Export

@BEG_Body

6

@BEG_Export

@BEG_Algo
@ALGORITHM @RT(12)aSensorState @STRUCTURED_TEXT
@RT(0) @RT(0) @RT(0) @F @F
@END_Algo

@BEG_Dcl
@RT(16)DclTreeContainer
0
@END_Dcl

@END_Export

@BEG_Export

@BEG_Algo
@PROCESS_ALGORITHM @RT(6)paInit @STRUCTURED_TEXT
@RT(0) @RT(0) @RT(8)TaskSlow @T @F
@END_Algo

@BEG_Dcl
@RT(16)DclTreeContainer
1
@Var @RT(8)swoState @RT(0) @T @T @DERIVED 0 @T @T @DT @RT(11)KSWO_Status @RT(0) @T @T @UNKNOWN 0 @F
@F @F
@T
@BEG_Attrib
3 @RT(0) @RT(0) @RT(0)
@END_Attrib
1 0 @F @F @F @F

@END_Dcl

@END_Export

@BEG_Export

@BEG_Algo
@PROCESS_ALGORITHM @RT(23)paHopperTempSupervision @STRUCTURED_TEXT
@RT(0) @RT(0) @RT(8)TaskSlow @F @F
@END_Algo

@BEG_Dcl
@RT(16)DclTreeContainer
4
@Var @RT(18)fbRTrigWarningTemp @RT(0) @T @T @DERIVED 0 @T @T @DT @RT(6)R_TRIG @RT(0) @T @T @UNKNOWN 0 @F
@F @F
@T
@BEG_Attrib
3 @RT(0) @RT(0) @RT(0)
@END_Attrib
1 0 @F @F @F @F

@Var @RT(16)fbRTrigAlarmTemp @RT(0) @T @T @DERIVED 0 @T @T @DT @RT(6)R_TRIG @RT(0) @T @T @UNKNOWN 0 @F
@F @F
@T
@BEG_Attrib
3 @RT(0) @RT(0) @RT(0)
@END_Attrib
1 0 @F @F @F @F

@Var @RT(20)fbRTrigWarningTempOk @RT(0) @T @T @DERIVED 0 @T @T @DT @RT(6)R_TRIG @RT(0) @T @T @UNKNOWN 0 @F
@F @F
@T
@BEG_Attrib
3 @RT(0) @RT(0) @RT(0)
@END_Attrib
1 0 @F @F @F @F

@Var @RT(18)fbRTrigAlarmTempOk @RT(0) @T @T @DERIVED 0 @T @T @DT @RT(6)R_TRIG @RT(0) @T @T @UNKNOWN 0 @F
@F @F
@T
@BEG_Attrib
3 @RT(0) @RT(0) @RT(0)
@END_Attrib
1 0 @F @F @F @F

@END_Dcl

@END_Export

@BEG_Export

@BEG_Algo
@PROCESS_ALGORITHM @RT(14)paHopperCooler @STRUCTURED_TEXT
@RT(0) @RT(0) @RT(8)TaskSlow @F @F
@END_Algo

@BEG_Dcl
@RT(16)DclTreeContainer
2
@Var @RT(19)fbRTrigStartCooling @RT(0) @T @T @DERIVED 0 @T @T @DT @RT(6)R_TRIG @RT(0) @T @T @UNKNOWN 0 @F
@F @F
@T
@BEG_Attrib
3 @RT(0) @RT(0) @RT(0)
@END_Attrib
1 0 @F @F @F @F

@Var @RT(18)fbRTrigStopCooling @RT(0) @T @T @DERIVED 0 @T @T @DT @RT(6)R_TRIG @RT(0) @T @T @UNKNOWN 0 @F
@F @F
@T
@BEG_Attrib
3 @RT(0) @RT(0) @RT(0)
@END_Attrib
1 0 @F @F @F @F

@END_Dcl

@END_Export

@BEG_Export

@BEG_Algo
@POSTUPDATE_ALGORITHM @RT(18)pSensorTypeChanged @STRUCTURED_TEXT
@RT(0) @RT(23)sv_HopperTempSensorType @RT(9)PU_Task_7 @F @F
@END_Algo

@BEG_Dcl
@RT(16)DclTreeContainer
0
@END_Dcl

@END_Export

@BEG_Export

@BEG_Algo
@POSTUPDATE_ALGORITHM @RT(19)pSensorStateChanged @STRUCTURED_TEXT
@RT(0) @RT(15)mpbSensorState^ @RT(9)PU_Task_7 @F @F
@END_Algo

@BEG_Dcl
@RT(16)DclTreeContainer
0
@END_Dcl

@END_Export

@BEG_Body
@TL(24)
(**************************************** WARNING ********************************************
 *** The KEBA Kemro K2 System including software is not intended for safety control tasks! ***
 ***                       For further information see Comment tab!                        ***
 *********************************************************************************************)

mbSensorError := ti_HopperTemp_stat;

IF mbSensorError THEN

   //reset digital output for cooling in case of sensor error
   IF IS_LINKED(do_HopperCooler) THEN
      do_HopperCooler := FALSE;
   END_IF;

   SET_ALARM(Name := erHopperTempSensor,
             SubID1 := sv_DeviceId.CompId,
             SubID2 := sv_DeviceId.IndexId,
             Param1 := msHWPath);
ELSE
   RESET_ALARM(Name := erHopperTempSensor,
               SubID1 := sv_DeviceId.CompId,
               SubID2 := sv_DeviceId.IndexId);
END_IF;

@END_Body

@@@BEG_Comment@@@
@TL(0)

@@@END_Comment@@@

@BEG_Body
@TL(30)
(**************************************** WARNING ********************************************
 *** The KEBA Kemro K2 System including software is not intended for safety control tasks! ***
 ***                       For further information see Comment tab!                        ***
 *********************************************************************************************)

IF IS_LINKED(ti_HopperTemp) AND IS_LINKED(ti_HopperTemp_stat) THEN

   ti_HopperTemp_sensor := sv_HopperTempSensorType;

   msHWPath := FGetHWPath(CONCAT(GET_MY_FU_NAME(),'.ti_HopperTemp'), TRUE);
   mpbSensorState := @ti_HopperTemp_stat;

   aSensorState();

   swoState := KSWO_AddVariable( Task := TaskSlow,
                                 Name := 'HopperTemperature',
                                 Variable := ti_HopperTemp);

   //start supervision of hopper temperature
   START_PROCESS_ALGORITHM(paHopperTempSupervision);

   IF IS_LINKED(do_HopperCooler) THEN
      //start algorithm for hopper cooling
      START_PROCESS_ALGORITHM(paHopperCooler);
   END_IF;
END_IF;

STOP_PROCESS_ALGORITHM();

@END_Body

@@@BEG_Comment@@@
@TL(1)
Check which Inputs and Outputs are available and start according process algorithms
@@@END_Comment@@@

@BEG_Body
@TL(39)
(**************************************** WARNING ********************************************
 *** The KEBA Kemro K2 System including software is not intended for safety control tasks! ***
 ***                       For further information see Comment tab!                        ***
 *********************************************************************************************)

fbRTrigWarningTemp(CLK := (ti_HopperTemp > sv_rWarnTemp));
fbRTrigWarningTempOk(CLK := (ti_HopperTemp < (sv_rWarnTemp - sv_rHopperTempHysteresis)));

fbRTrigAlarmTemp(CLK := (ti_HopperTemp > sv_rAlarmTemp));
fbRTrigAlarmTempOk(CLK := (ti_HopperTemp < (sv_rAlarmTemp - sv_rHopperTempHysteresis)));

IF fbRTrigWarningTemp.Q THEN
   //set alarm if warning temp is exceeded
   SET_ALARM (Name := erHopperTempWarning,
              SubID1 := sv_DeviceId.CompId,
              SubID2 := sv_DeviceId.IndexId);
END_IF;

IF fbRTrigWarningTempOk.Q THEN
   //reset alarm if temp is ok again
   RESET_ALARM (Name := erHopperTempWarning,
                SubID1 := sv_DeviceId.CompId,
                SubID2 := sv_DeviceId.IndexId);
END_IF;

IF fbRTrigAlarmTemp.Q THEN
   //set alarm if alarm temp is exceeded
   SET_ALARM (Name := erHopperTempTooHigh,
              SubID1 := sv_DeviceId.CompId,
              SubID2 := sv_DeviceId.IndexId);
END_IF;

IF fbRTrigAlarmTempOk.Q THEN
   //set alarm if temp is ok again
   RESET_ALARM (Name := erHopperTempTooHigh,
                SubID1 := sv_DeviceId.CompId,
                SubID2 := sv_DeviceId.IndexId);
END_IF;

@END_Body

@@@BEG_Comment@@@
@TL(5)
In this algorithm the supervision of the material temperature is done.
If actual material temp is higher than the alarm temperature an alarm is set.
If actual material temperature is lower than alarm temp -5° the alarm is resetted.
Setting the material temp high - alarm causes a stop of the motor!
Switching on the motor is only possible if the material temperature is ok again.
@@@END_Comment@@@

@BEG_Body
@TL(20)
(**************************************** WARNING ********************************************
 *** The KEBA Kemro K2 System including software is not intended for safety control tasks! ***
 ***                       For further information see Comment tab!                        ***
 *********************************************************************************************)

fbRTrigStartCooling(CLK := (ti_HopperTemp > sv_rTempStartCooling));
fbRTrigStopCooling(CLK := (ti_HopperTemp < sv_rTempStopCooling));

IF fbRTrigStartCooling.Q AND NOT mbSensorError THEN
   //set digital output for cooling
   do_HopperCooler := TRUE;
END_IF;

IF fbRTrigStopCooling.Q THEN
   //reset digital output for cooling
   do_HopperCooler := FALSE;
END_IF;

@END_Body

@@@BEG_Comment@@@
@TL(4)
If a digital output for hopper cooling is available it will be set if the
actual material temperature is higher than start cooling temperature.
The DO will be resetted after the actual temperature is lower than stop cooling temperature.
In case of a sensor error the DO will also be resetted.
@@@END_Comment@@@

@BEG_Body
@TL(9)
(**************************************** WARNING ********************************************
 *** The KEBA Kemro K2 System including software is not intended for safety control tasks! ***
 ***                       For further information see Comment tab!                        ***
 *********************************************************************************************)

//copy selected sensor type
ti_HopperTemp_sensor := sv_HopperTempSensorType;

@END_Body

@@@BEG_Comment@@@
@TL(0)

@@@END_Comment@@@

@BEG_Body
@TL(9)
(**************************************** WARNING ********************************************
 *** The KEBA Kemro K2 System including software is not intended for safety control tasks! ***
 ***                       For further information see Comment tab!                        ***
 *********************************************************************************************)

aSensorState();

@END_Body

@@@BEG_Comment@@@
@TL(1)
react on changes of material temp sensor state
@@@END_Comment@@@
@END_Body

@END_Contents
